FUNCTION_BLOCK BIT_TO_INT (* Basic Function Block Type *)
  (* Standard: 61499-2 *)
  (* Version 0.0, 30/11/2020, Schulung, Schneider Electric, Template *)
  PACKAGE Main;
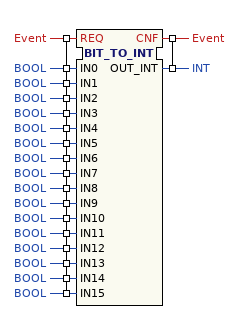
  EVENT_INPUT
    REQ WITH IN0, IN1, IN2, IN3, IN4, IN5, IN6, IN7, IN8, IN9, IN10, IN11, IN12, IN13, IN14, IN15; (* Normal Execution Request *)
  END_EVENT
  EVENT_OUTPUT
    CNF WITH OUT_INT; (* Execution Confirmation *)
  END_EVENT
  VAR_INPUT
    IN0 : BOOL; (* Input event qualifier *)
    IN1 : BOOL;
    IN2 : BOOL;
    IN3 : BOOL;
    IN4 : BOOL;
    IN5 : BOOL;
    IN6 : BOOL;
    IN7 : BOOL;
    IN8 : BOOL;
    IN9 : BOOL;
    IN10 : BOOL;
    IN11 : BOOL;
    IN12 : BOOL;
    IN13 : BOOL;
    IN14 : BOOL;
    IN15 : BOOL;
  END_VAR
  VAR_OUTPUT
    OUT_INT : INT; (* Output event qualifier *)
  END_VAR
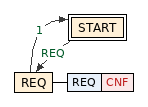
  EC_STATES
    START; (* Initial State *)
    REQ : REQ -> CNF; (* Normal execution *)
  END_STATES
  EC_TRANSITIONS
    START TO REQ := REQ;
    REQ TO START := 1;
  END_TRANSITIONS
  ALGORITHM REQ IN ST: (* Normally executed algorithm *)
OUT_INT :=
	WORD_TO_INT(SHL(BOOL_TO_WORD(IN0),0)
	+ SHL(BOOL_TO_WORD(IN1),1)
	+ SHL(BOOL_TO_WORD(IN2),2)
	+ SHL(BOOL_TO_WORD(IN3),3)
	+ SHL(BOOL_TO_WORD(IN4),4)
	+ SHL(BOOL_TO_WORD(IN5),5)
	+ SHL(BOOL_TO_WORD(IN6),6)
	+ SHL(BOOL_TO_WORD(IN7),7)
	+ SHL(BOOL_TO_WORD(IN8),8)
	+ SHL(BOOL_TO_WORD(IN9),9)
	+ SHL(BOOL_TO_WORD(IN10),10)
	+ SHL(BOOL_TO_WORD(IN11),11)
	+ SHL(BOOL_TO_WORD(IN12),12)
	+ SHL(BOOL_TO_WORD(IN13),13)
	+ SHL(BOOL_TO_WORD(IN14),14)
	+ SHL(BOOL_TO_WORD(IN15),15))
	;
  END_ALGORITHM
END_FUNCTION_BLOCK
